// TIA Portal V18 export
ORGANIZATION_BLOCK "Main"   // OB123, FBD, ProgramCycle
TITLE = "Main Program Sweep (Cycle)"
{ S7_Optimized_Access := 'TRUE' }
VERSION : 0.1
// stored: AutoNumber true, IsIECCheckEnabled false, SetENOAutomatically false
   VAR_INPUT
      Initial_Call : Bool;   // Initial call of this OB
      Remanence : Bool;   // =True, if remanent data are available
   END_VAR
BEGIN

REGION Network 1 (SCL): HSSR_019 SOURCE SELECTION

   "Source_select_H/SSR_019_DB".START := "H/SSR_019_START";
   "Source_select_H/SSR_019_DB".SP := "H/SSR_019_SP";
   "Source_select_H/SSR_019_DB".PV := "H/SSR_019_TT01_PV";
   "Source_select_H/SSR_019_DB".COUNTER_SP := "H/SSR_019_ALERT_SP";
   "Source_select_H/SSR_019_DB".CHW_CT_SP := "H/SSR_019_CHBr_RT_SP";
   "Source_select_H/SSR_019_DB".CT_HW_SP := "H/SSR_019_RT_HW_SP";
   "Source_select_H/SSR_019_DB".HW_STEAM_SP := "H/SSR_019_HW_STEAM_SP";
   "Source_select_H/SSR_019_DB".CT_CHW_SP := "H/SSR_019_RT_CHBr_SP";

   "H/SSR_019_SOURCE_SEL" := "Source_select_H/SSR_019_DB".SOURCE_SEL;
END_REGION

REGION Network 2 (SCL): HSSR_019 UTILITY PID

   "Utility_PID_DB".AM := "H/SSR_019_AM";
   "Utility_PID_DB".START := "H/SSR_019_START";
   "Utility_PID_DB".SP := "H/SSR_019_SP";
   "Utility_PID_DB".PV := "H/SSR_019_TT01_PV";
   "Utility_PID_DB".TIME := "H/SSR_019_TIME_SP";
   "Utility_PID_DB".P := "H/SSR_019_KP";
   "Utility_PID_DB".I := "H/SSR_019_TI";
   "Utility_PID_DB".JAC_IN := "H/SSR_019_TT02_PV";
   "Utility_PID_DB".SOURCE_SEL := "Source_select_H/SSR_019_DB".SOURCE_SEL;
   "Utility_PID_DB".MAN_OUT := "H/SSR_019_CV02_MANOUT";
   "Utility_PID_DB".STEAM_MAN_OUT := "H/SSR_019_CV01_MANOUT";
   "Utility_PID_DB".AIR_XV_OPN := "H/SSR_019_XV10_CMD";
   "Utility_PID_DB".BYP_XV_OPN := "H/SSR_019_XV05_CMD";
   "Utility_PID_DB".VENT_OPN := "H/SSR_019_XV06_CMD";
   "Utility_PID_DB".CONDENSATE_XV_OPN := "H/SSR_019_XV12_CMD";
   "Utility_PID_DB".DRAIN_XV_OPN := "H/SSR_019_XV13_CMD";
   "Utility_PID_DB".CONTROL_MODE := 1;

   "H/SSR_019_START_PV" := "Utility_PID_DB".START_PV;
   "H/SSR_019_CV02_SCVOUT" := "Utility_PID_DB".SCVOUT;
   "H/SSR_019_CV02_CVOUT" := "Utility_PID_DB".CVOUT;
   "H/SSR_019_CV01_SCVOUT" := "Utility_PID_DB".STEAM_SCVOUT;
   "H/SSR_019_CV01_CVOUT" := "Utility_PID_DB".STEAM_CVOUT;
   "H/SSR_019_RUN_MIN" := "Utility_PID_DB".RUN_MIN;
END_REGION

REGION Network 3 (SCL): HSSR_019 UTILITY SELECTION

   "Utility_selection_DB".utl_type :=  "Source_select_H/SSR_019_DB".SOURCE_SEL;
   "Utility_selection_DB".chws_cfb :="SIM_VALVE"."H/SSR_019_XV01_CLOSEFB" ;
   "Utility_selection_DB".chws_ofb := "SIM_VALVE"."H/SSR_019_XV01_OPENFB";
   "Utility_selection_DB".cws_cfb := "SIM_VALVE"."H/SSR_019_XV02_CLOSEFB";
   "Utility_selection_DB".cws_ofb := "SIM_VALVE"."H/SSR_019_XV02_OPENFB";
   "Utility_selection_DB".hws_cfb := "SIM_VALVE"."H/SSR_019_XV03_CLOSEFB";
   "Utility_selection_DB".hws_ofb := "SIM_VALVE"."H/SSR_019_XV03_OPENFB";
   "Utility_selection_DB".chwr_cfb := "SIM_VALVE"."H/SSR_019_XV07_CLOSEFB";
   "Utility_selection_DB".chwr_ofb := "SIM_VALVE"."H/SSR_019_XV07_OPENFB";
   "Utility_selection_DB".cwr_cfb := "SIM_VALVE"."H/SSR_019_XV08_CLOSEFB";
   "Utility_selection_DB".cwr_ofb := "SIM_VALVE"."H/SSR_019_XV08_OPENFB";
   "Utility_selection_DB".hwr_cfb := "SIM_VALVE"."H/SSR_019_XV09_CLOSEFB";
   "Utility_selection_DB".hwr_ofb := "SIM_VALVE"."H/SSR_019_XV09_OPENFB";
   "Utility_selection_DB".scv_ofb := "SIM_VALVE"."H/SSR_019_XV11_OPENFB";
   "Utility_selection_DB".cond_cfb := "SIM_VALVE"."H/SSR_019_XV12_CLOSEFB";
   "Utility_selection_DB".cond_ofb := "SIM_VALVE"."H/SSR_019_XV12_OPENFB";
   "Utility_selection_DB".dr_cfb := "SIM_VALVE"."H/SSR_019_XV13_CLOSEFB";
   "Utility_selection_DB".dr_ofb := "SIM_VALVE"."H/SSR_019_XV13_OPENFB";
   "Utility_selection_DB".as_cfb := "SIM_VALVE"."H/SSR_019_XV10_CLOSEFB";
   "Utility_selection_DB".as_ofb := "SIM_VALVE"."H/SSR_019_XV10_OPENFB";
   "Utility_selection_DB".av_cfb := "SIM_VALVE"."H/SSR_019_XV06_CLOSEFB";
   "Utility_selection_DB".av_ofb := "SIM_VALVE"."H/SSR_019_XV06_OPENFB";
   "Utility_selection_DB".utl_bit := "H/SSR_019_START";
   "Utility_selection_DB".control.%X1 := "H/SSR_019_AM";
   "Utility_selection_DB".control.%X2 := "H/SSR_019_START";
   "Utility_selection_DB".times[0] := "H/SSR_019_FLUSH_TIME_SP";
   "Utility_selection_DB".times[1] := "H/SSR_019_VENT_TIME_SP";
   "Utility_selection_DB".times[2] := "H/SSR_019_CONDENSATE_TIME_SP";
   "Utility_selection_DB".control.%X0   := "H/SSR_019_HOLD";
   "Utility_selection_DB".control.%X6 := "H/SSR_019_EMSTOP";
   "Utility_selection_DB".byp_cfb := "SIM_VALVE"."H/SSR_019_XV05_CLOSEFB";
   "Utility_selection_DB".byp_ofb := "SIM_VALVE"."H/SSR_019_XV05_OPENFB";
   "H/SSR_019_XV01_CMD" := "Utility_selection_DB".chws_cmd;
   "H/SSR_019_XV02_CMD" := "Utility_selection_DB".cws_cmd;
   "H/SSR_019_XV03_CMD" := "Utility_selection_DB".hws_cmd;
   "H/SSR_019_XV07_CMD" := "Utility_selection_DB".chwr_cmd;
   "H/SSR_019_XV08_CMD" := "Utility_selection_DB".cwr_cmd;
   "H/SSR_019_XV09_CMD" := "Utility_selection_DB".hwr_cmd;
   "H/SSR_019_XV11_CMD" := "Utility_selection_DB".scv_cmd;
   "H/SSR_019_XV12_CMD" := "Utility_selection_DB".cond_cmd;
   "H/SSR_019_XV13_CMD" := "Utility_selection_DB".dr_cmd;
   "H/SSR_019_XV10_CMD" := "Utility_selection_DB".as_cmd;
   "H/SSR_019_XV05_CMD" := "Utility_selection_DB".byp_cmd;
   "H/SSR_019_XV06_CMD" := "Utility_selection_DB".av_cmd;
   "H/SSR_019_FLUSH_RUN_TIME" := "Utility_selection_DB".flush_time;
   "H/SSR_019_CONDENSATE_RUN_TIME" := "Utility_selection_DB".drine_time;
   "H/SSR_019_VENT_RUN_TIME" := "Utility_selection_DB".vent_time;
   "H/SSR_019_Flush_CMP" := "Utility_selection_DB".status.%X2;
   "H/SSR_019_Vent_CMP" := "Utility_selection_DB".status.%X3;
   "H/SSR_019_Cond_CMP" := "Utility_selection_DB".status.%X4;
END_REGION

REGION Network 4: HSSR_019_Pre checks
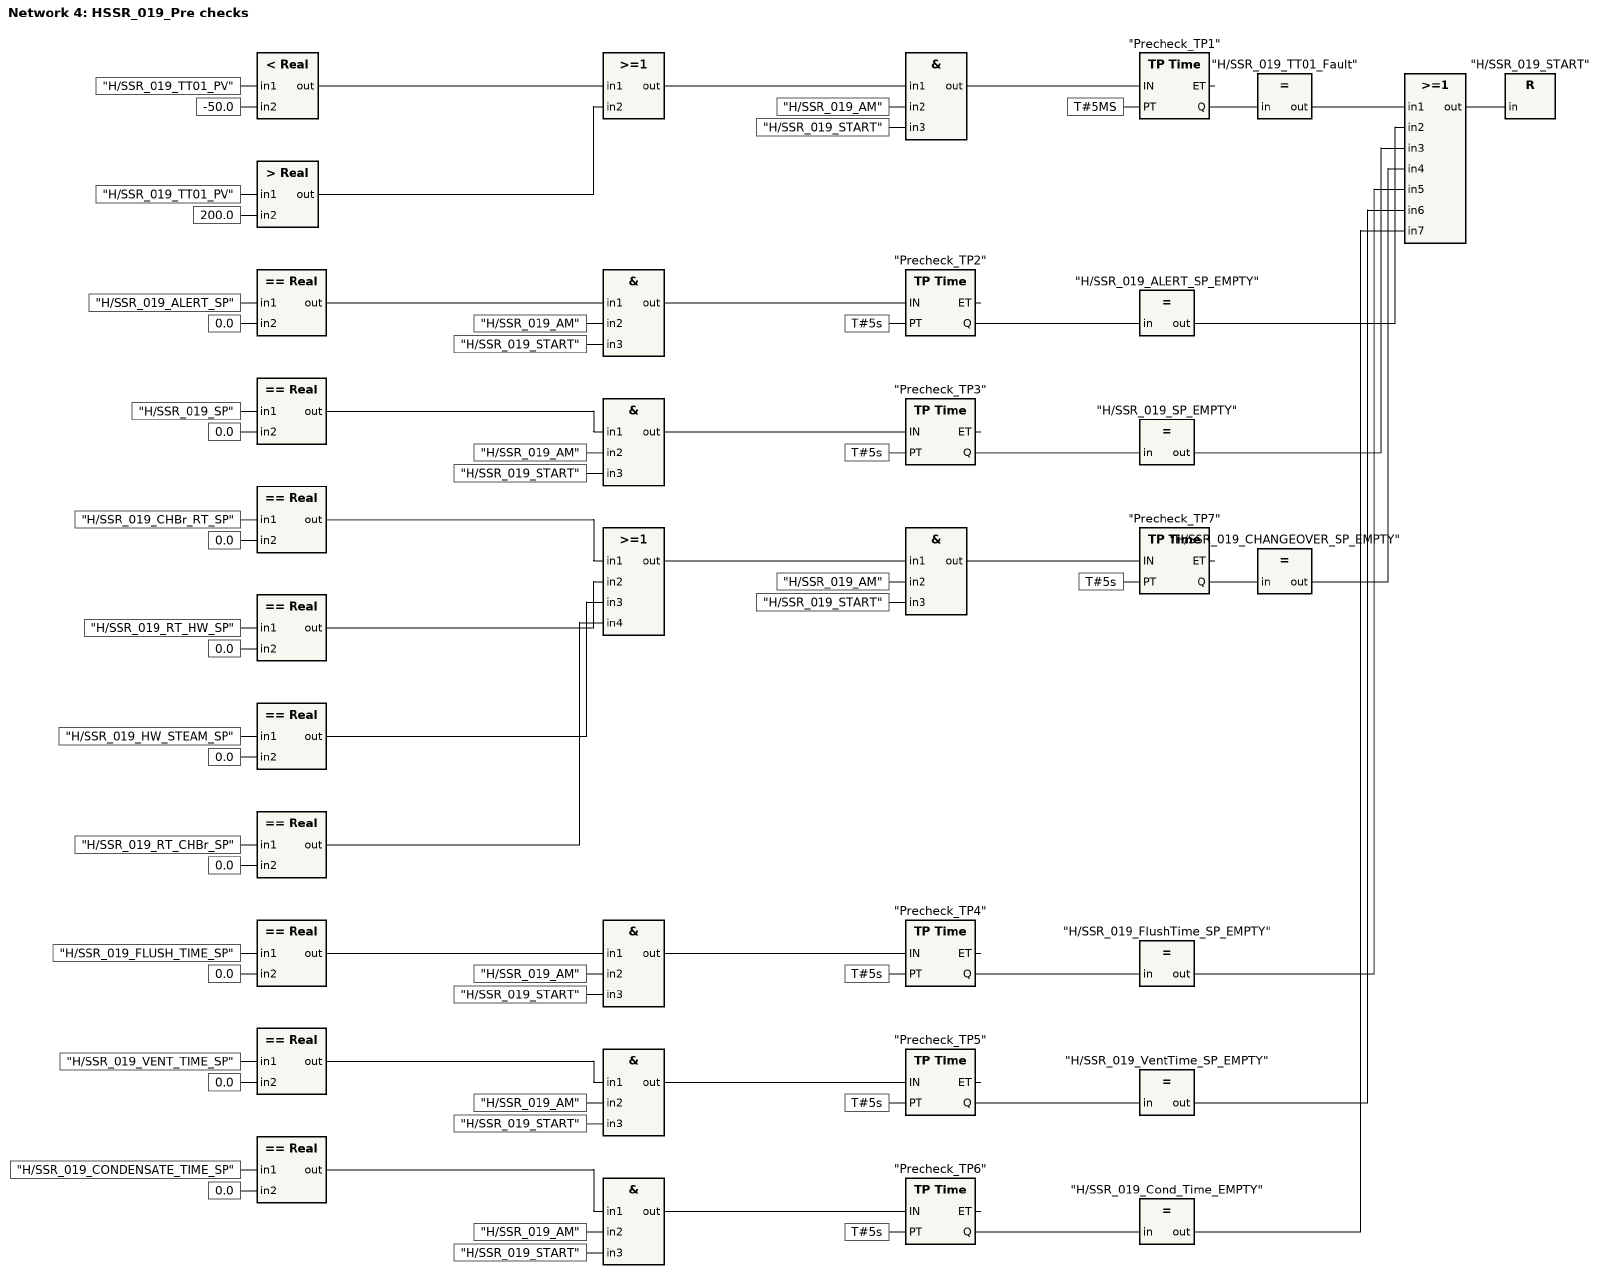
   "Precheck_TP1".TP(IN := (("H/SSR_019_TT01_PV" < (-50.0)) OR ("H/SSR_019_TT01_PV" > 200.0)) AND "H/SSR_019_AM" AND "H/SSR_019_START",
                     PT := T#5MS);
   "H/SSR_019_TT01_Fault" := "Precheck_TP1".Q;
   "Precheck_TP2".TP(IN := ("H/SSR_019_ALERT_SP" = 0.0) AND "H/SSR_019_AM" AND "H/SSR_019_START", PT := T#5s);
   "H/SSR_019_ALERT_SP_EMPTY" := "Precheck_TP2".Q;
   "Precheck_TP3".TP(IN := ("H/SSR_019_SP" = 0.0) AND "H/SSR_019_AM" AND "H/SSR_019_START", PT := T#5s);
   "H/SSR_019_SP_EMPTY" := "Precheck_TP3".Q;
   "Precheck_TP7".TP(IN := (("H/SSR_019_CHBr_RT_SP" = 0.0) OR ("H/SSR_019_RT_HW_SP" = 0.0) OR ("H/SSR_019_HW_STEAM_SP" = 0.0) OR ("H/SSR_019_RT_CHBr_SP" = 0.0)) AND "H/SSR_019_AM" AND "H/SSR_019_START",
                     PT := T#5s);
   "H/SSR_019_CHANGEOVER_SP_EMPTY" := "Precheck_TP7".Q;
   "Precheck_TP4".TP(IN := ("H/SSR_019_FLUSH_TIME_SP" = 0.0) AND "H/SSR_019_AM" AND "H/SSR_019_START",
                     PT := T#5s);
   "H/SSR_019_FlushTime_SP_EMPTY" := "Precheck_TP4".Q;
   "Precheck_TP5".TP(IN := ("H/SSR_019_VENT_TIME_SP" = 0.0) AND "H/SSR_019_AM" AND "H/SSR_019_START",
                     PT := T#5s);
   "H/SSR_019_VentTime_SP_EMPTY" := "Precheck_TP5".Q;
   "Precheck_TP6".TP(IN := ("H/SSR_019_CONDENSATE_TIME_SP" = 0.0) AND "H/SSR_019_AM" AND "H/SSR_019_START",
                     PT := T#5s);
   "H/SSR_019_Cond_Time_EMPTY" := "Precheck_TP6".Q;
   IF "Precheck_TP1".Q OR "Precheck_TP2".Q OR "Precheck_TP3".Q OR "Precheck_TP7".Q OR "Precheck_TP4".Q OR "Precheck_TP5".Q OR "Precheck_TP6".Q THEN
       "H/SSR_019_START" := FALSE;
   END_IF;
END_REGION

REGION Network 5: H/SSR_019Valves
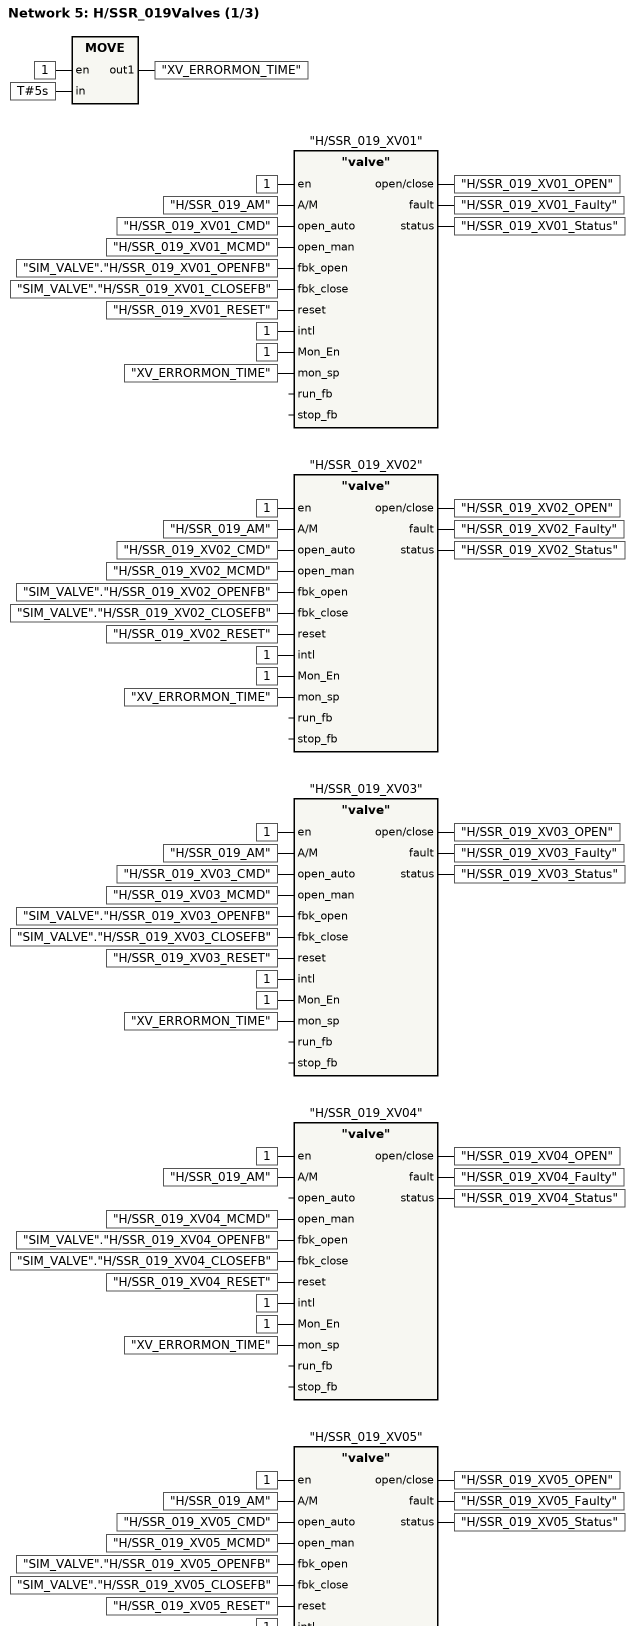
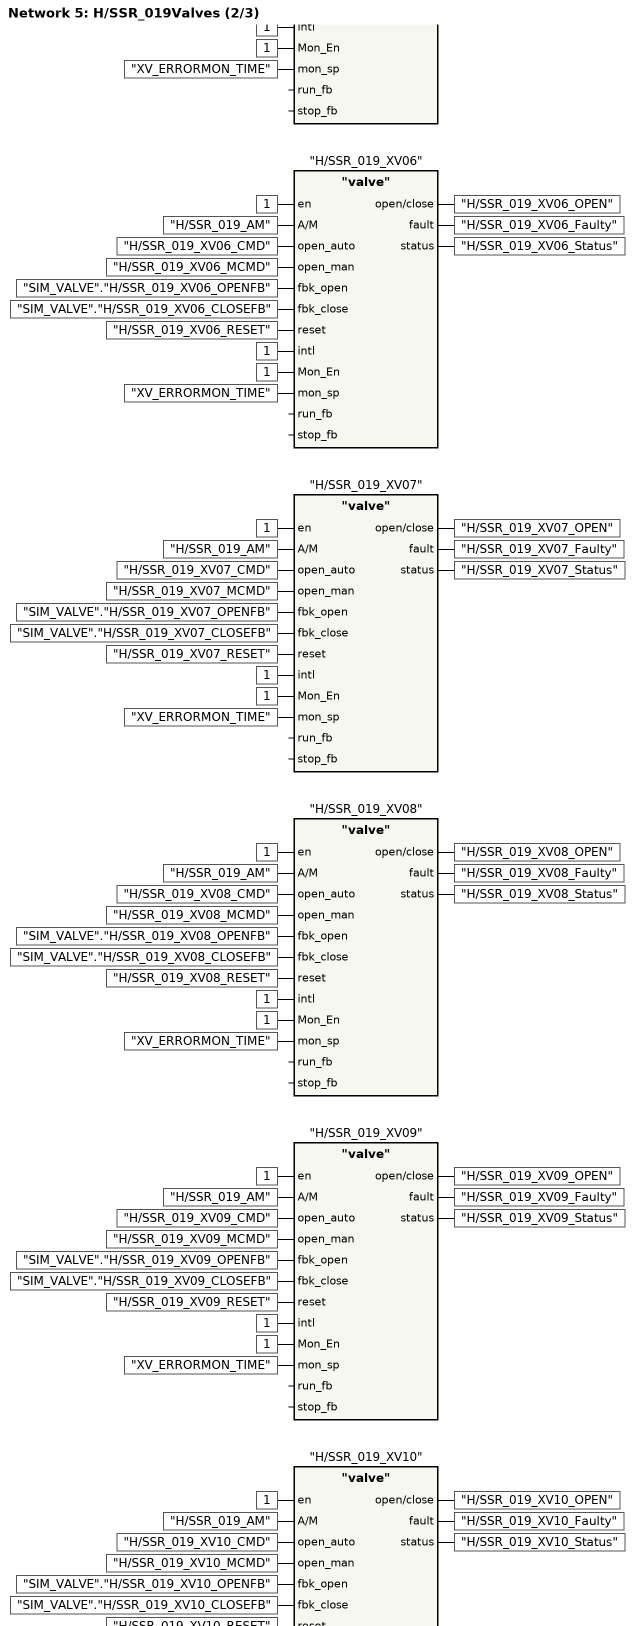
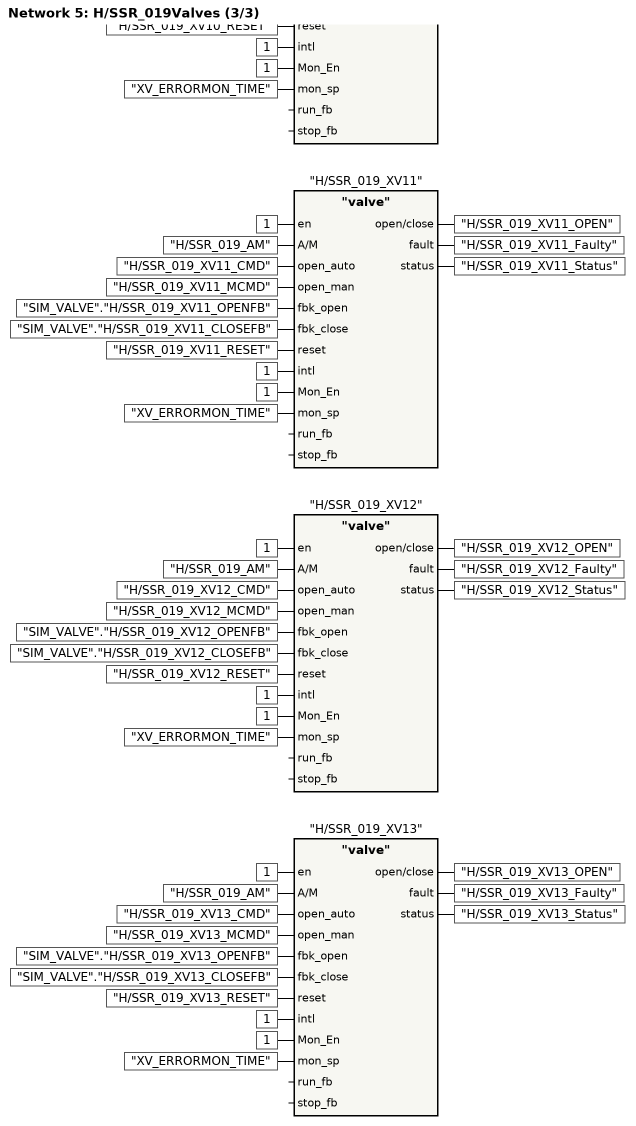
   IF 1 THEN
       "XV_ERRORMON_TIME" := T#5s;
       "H/SSR_019_XV01"("A/M" := "H/SSR_019_AM",   // "valve"
                        open_auto := "H/SSR_019_XV01_CMD",
                        open_man := "H/SSR_019_XV01_MCMD",
                        fbk_open := "SIM_VALVE"."H/SSR_019_XV01_OPENFB",
                        fbk_close := "SIM_VALVE"."H/SSR_019_XV01_CLOSEFB",
                        reset := "H/SSR_019_XV01_RESET",
                        intl := 1,
                        Mon_En := 1,
                        mon_sp := "XV_ERRORMON_TIME",
                        "open/close" => "H/SSR_019_XV01_OPEN",
                        fault => "H/SSR_019_XV01_Faulty",
                        status => "H/SSR_019_XV01_Status");
       "H/SSR_019_XV02"("A/M" := "H/SSR_019_AM",   // "valve"
                        open_auto := "H/SSR_019_XV02_CMD",
                        open_man := "H/SSR_019_XV02_MCMD",
                        fbk_open := "SIM_VALVE"."H/SSR_019_XV02_OPENFB",
                        fbk_close := "SIM_VALVE"."H/SSR_019_XV02_CLOSEFB",
                        reset := "H/SSR_019_XV02_RESET",
                        intl := 1,
                        Mon_En := 1,
                        mon_sp := "XV_ERRORMON_TIME",
                        "open/close" => "H/SSR_019_XV02_OPEN",
                        fault => "H/SSR_019_XV02_Faulty",
                        status => "H/SSR_019_XV02_Status");
       "H/SSR_019_XV03"("A/M" := "H/SSR_019_AM",   // "valve"
                        open_auto := "H/SSR_019_XV03_CMD",
                        open_man := "H/SSR_019_XV03_MCMD",
                        fbk_open := "SIM_VALVE"."H/SSR_019_XV03_OPENFB",
                        fbk_close := "SIM_VALVE"."H/SSR_019_XV03_CLOSEFB",
                        reset := "H/SSR_019_XV03_RESET",
                        intl := 1,
                        Mon_En := 1,
                        mon_sp := "XV_ERRORMON_TIME",
                        "open/close" => "H/SSR_019_XV03_OPEN",
                        fault => "H/SSR_019_XV03_Faulty",
                        status => "H/SSR_019_XV03_Status");
       "H/SSR_019_XV04"("A/M" := "H/SSR_019_AM",   // "valve"
                        open_man := "H/SSR_019_XV04_MCMD",
                        fbk_open := "SIM_VALVE"."H/SSR_019_XV04_OPENFB",
                        fbk_close := "SIM_VALVE"."H/SSR_019_XV04_CLOSEFB",
                        reset := "H/SSR_019_XV04_RESET",
                        intl := 1,
                        Mon_En := 1,
                        mon_sp := "XV_ERRORMON_TIME",
                        "open/close" => "H/SSR_019_XV04_OPEN",
                        fault => "H/SSR_019_XV04_Faulty",
                        status => "H/SSR_019_XV04_Status");
       "H/SSR_019_XV05"("A/M" := "H/SSR_019_AM",   // "valve"
                        open_auto := "H/SSR_019_XV05_CMD",
                        open_man := "H/SSR_019_XV05_MCMD",
                        fbk_open := "SIM_VALVE"."H/SSR_019_XV05_OPENFB",
                        fbk_close := "SIM_VALVE"."H/SSR_019_XV05_CLOSEFB",
                        reset := "H/SSR_019_XV05_RESET",
                        intl := 1,
                        Mon_En := 1,
                        mon_sp := "XV_ERRORMON_TIME",
                        "open/close" => "H/SSR_019_XV05_OPEN",
                        fault => "H/SSR_019_XV05_Faulty",
                        status => "H/SSR_019_XV05_Status");
       "H/SSR_019_XV06"("A/M" := "H/SSR_019_AM",   // "valve"
                        open_auto := "H/SSR_019_XV06_CMD",
                        open_man := "H/SSR_019_XV06_MCMD",
                        fbk_open := "SIM_VALVE"."H/SSR_019_XV06_OPENFB",
                        fbk_close := "SIM_VALVE"."H/SSR_019_XV06_CLOSEFB",
                        reset := "H/SSR_019_XV06_RESET",
                        intl := 1,
                        Mon_En := 1,
                        mon_sp := "XV_ERRORMON_TIME",
                        "open/close" => "H/SSR_019_XV06_OPEN",
                        fault => "H/SSR_019_XV06_Faulty",
                        status => "H/SSR_019_XV06_Status");
       "H/SSR_019_XV07"("A/M" := "H/SSR_019_AM",   // "valve"
                        open_auto := "H/SSR_019_XV07_CMD",
                        open_man := "H/SSR_019_XV07_MCMD",
                        fbk_open := "SIM_VALVE"."H/SSR_019_XV07_OPENFB",
                        fbk_close := "SIM_VALVE"."H/SSR_019_XV07_CLOSEFB",
                        reset := "H/SSR_019_XV07_RESET",
                        intl := 1,
                        Mon_En := 1,
                        mon_sp := "XV_ERRORMON_TIME",
                        "open/close" => "H/SSR_019_XV07_OPEN",
                        fault => "H/SSR_019_XV07_Faulty",
                        status => "H/SSR_019_XV07_Status");
       "H/SSR_019_XV08"("A/M" := "H/SSR_019_AM",   // "valve"
                        open_auto := "H/SSR_019_XV08_CMD",
                        open_man := "H/SSR_019_XV08_MCMD",
                        fbk_open := "SIM_VALVE"."H/SSR_019_XV08_OPENFB",
                        fbk_close := "SIM_VALVE"."H/SSR_019_XV08_CLOSEFB",
                        reset := "H/SSR_019_XV08_RESET",
                        intl := 1,
                        Mon_En := 1,
                        mon_sp := "XV_ERRORMON_TIME",
                        "open/close" => "H/SSR_019_XV08_OPEN",
                        fault => "H/SSR_019_XV08_Faulty",
                        status => "H/SSR_019_XV08_Status");
       "H/SSR_019_XV09"("A/M" := "H/SSR_019_AM",   // "valve"
                        open_auto := "H/SSR_019_XV09_CMD",
                        open_man := "H/SSR_019_XV09_MCMD",
                        fbk_open := "SIM_VALVE"."H/SSR_019_XV09_OPENFB",
                        fbk_close := "SIM_VALVE"."H/SSR_019_XV09_CLOSEFB",
                        reset := "H/SSR_019_XV09_RESET",
                        intl := 1,
                        Mon_En := 1,
                        mon_sp := "XV_ERRORMON_TIME",
                        "open/close" => "H/SSR_019_XV09_OPEN",
                        fault => "H/SSR_019_XV09_Faulty",
                        status => "H/SSR_019_XV09_Status");
       "H/SSR_019_XV10"("A/M" := "H/SSR_019_AM",   // "valve"
                        open_auto := "H/SSR_019_XV10_CMD",
                        open_man := "H/SSR_019_XV10_MCMD",
                        fbk_open := "SIM_VALVE"."H/SSR_019_XV10_OPENFB",
                        fbk_close := "SIM_VALVE"."H/SSR_019_XV10_CLOSEFB",
                        reset := "H/SSR_019_XV10_RESET",
                        intl := 1,
                        Mon_En := 1,
                        mon_sp := "XV_ERRORMON_TIME",
                        "open/close" => "H/SSR_019_XV10_OPEN",
                        fault => "H/SSR_019_XV10_Faulty",
                        status => "H/SSR_019_XV10_Status");
       "H/SSR_019_XV11"("A/M" := "H/SSR_019_AM",   // "valve"
                        open_auto := "H/SSR_019_XV11_CMD",
                        open_man := "H/SSR_019_XV11_MCMD",
                        fbk_open := "SIM_VALVE"."H/SSR_019_XV11_OPENFB",
                        fbk_close := "SIM_VALVE"."H/SSR_019_XV11_CLOSEFB",
                        reset := "H/SSR_019_XV11_RESET",
                        intl := 1,
                        Mon_En := 1,
                        mon_sp := "XV_ERRORMON_TIME",
                        "open/close" => "H/SSR_019_XV11_OPEN",
                        fault => "H/SSR_019_XV11_Faulty",
                        status => "H/SSR_019_XV11_Status");
       "H/SSR_019_XV12"("A/M" := "H/SSR_019_AM",   // "valve"
                        open_auto := "H/SSR_019_XV12_CMD",
                        open_man := "H/SSR_019_XV12_MCMD",
                        fbk_open := "SIM_VALVE"."H/SSR_019_XV12_OPENFB",
                        fbk_close := "SIM_VALVE"."H/SSR_019_XV12_CLOSEFB",
                        reset := "H/SSR_019_XV12_RESET",
                        intl := 1,
                        Mon_En := 1,
                        mon_sp := "XV_ERRORMON_TIME",
                        "open/close" => "H/SSR_019_XV12_OPEN",
                        fault => "H/SSR_019_XV12_Faulty",
                        status => "H/SSR_019_XV12_Status");
       "H/SSR_019_XV13"("A/M" := "H/SSR_019_AM",   // "valve"
                        open_auto := "H/SSR_019_XV13_CMD",
                        open_man := "H/SSR_019_XV13_MCMD",
                        fbk_open := "SIM_VALVE"."H/SSR_019_XV13_OPENFB",
                        fbk_close := "SIM_VALVE"."H/SSR_019_XV13_CLOSEFB",
                        reset := "H/SSR_019_XV13_RESET",
                        intl := 1,
                        Mon_En := 1,
                        mon_sp := "XV_ERRORMON_TIME",
                        "open/close" => "H/SSR_019_XV13_OPEN",
                        fault => "H/SSR_019_XV13_Faulty",
                        status => "H/SSR_019_XV13_Status");
   END_IF;
END_REGION

REGION Network 6: AI_H/SSR_019_ Reading
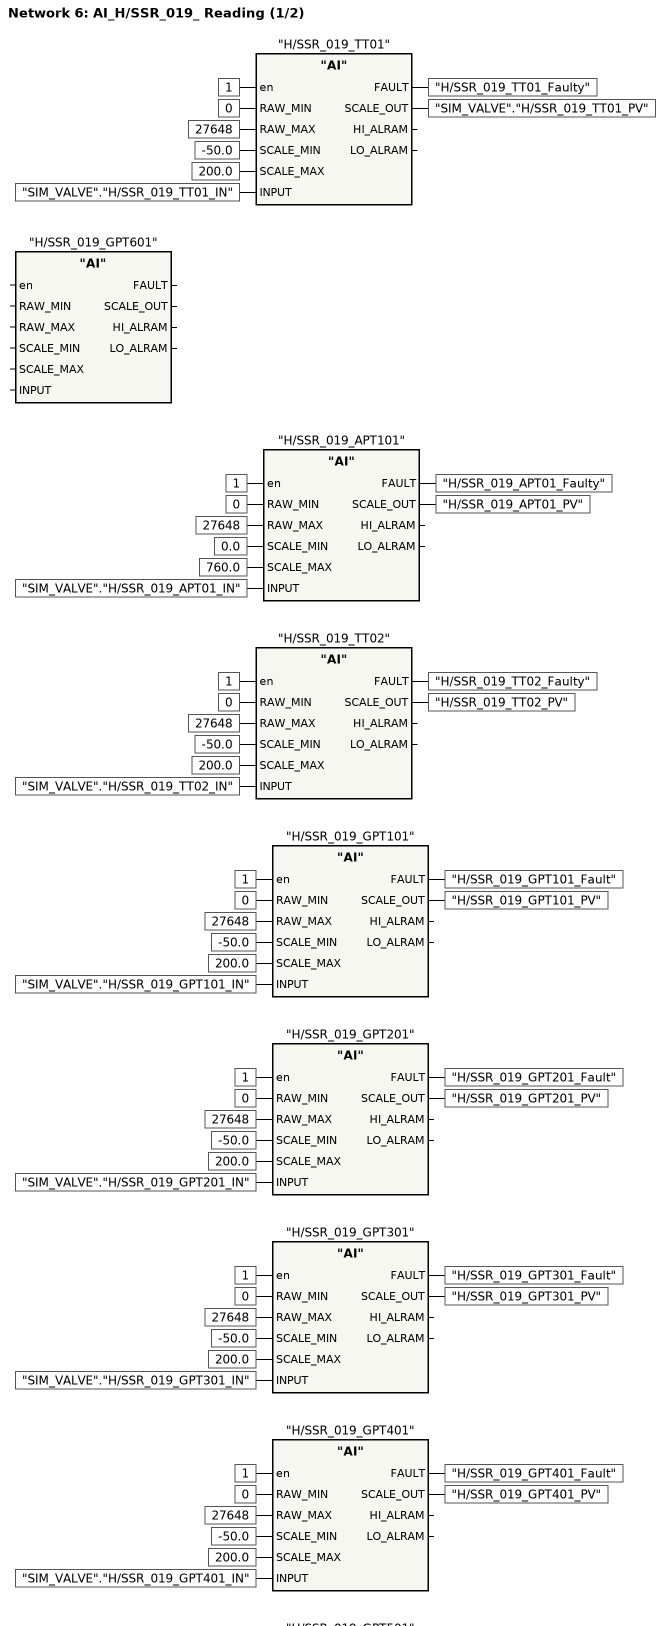
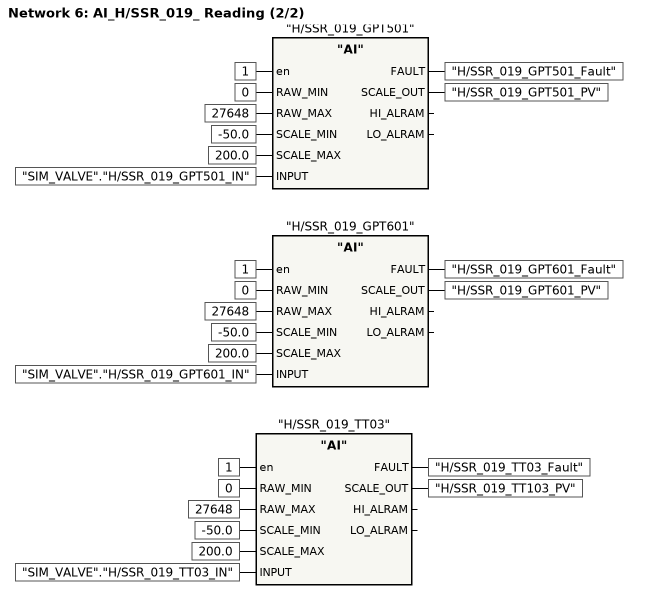
   IF 1 THEN
       "H/SSR_019_TT01"(RAW_MIN := 0,   // "AI"
                        RAW_MAX := 27648,
                        SCALE_MIN := -50.0,
                        SCALE_MAX := 200.0,
                        INPUT := "SIM_VALVE"."H/SSR_019_TT01_IN",
                        FAULT => "H/SSR_019_TT01_Faulty",
                        SCALE_OUT => "SIM_VALVE"."H/SSR_019_TT01_PV");
   END_IF;
   "H/SSR_019_GPT601"();   // "AI"
   IF 1 THEN
       "H/SSR_019_APT101"(RAW_MIN := 0,   // "AI"
                          RAW_MAX := 27648,
                          SCALE_MIN := 0.0,
                          SCALE_MAX := 760.0,
                          INPUT := "SIM_VALVE"."H/SSR_019_APT01_IN",
                          FAULT => "H/SSR_019_APT01_Faulty",
                          SCALE_OUT => "H/SSR_019_APT01_PV");
       "H/SSR_019_TT02"(RAW_MIN := 0,   // "AI"
                        RAW_MAX := 27648,
                        SCALE_MIN := -50.0,
                        SCALE_MAX := 200.0,
                        INPUT := "SIM_VALVE"."H/SSR_019_TT02_IN",
                        FAULT => "H/SSR_019_TT02_Faulty",
                        SCALE_OUT => "H/SSR_019_TT02_PV");
       "H/SSR_019_GPT101"(RAW_MIN := 0,   // "AI"
                          RAW_MAX := 27648,
                          SCALE_MIN := -50.0,
                          SCALE_MAX := 200.0,
                          INPUT := "SIM_VALVE"."H/SSR_019_GPT101_IN",
                          FAULT => "H/SSR_019_GPT101_Fault",
                          SCALE_OUT => "H/SSR_019_GPT101_PV");
       "H/SSR_019_GPT201"(RAW_MIN := 0,   // "AI"
                          RAW_MAX := 27648,
                          SCALE_MIN := -50.0,
                          SCALE_MAX := 200.0,
                          INPUT := "SIM_VALVE"."H/SSR_019_GPT201_IN",
                          FAULT => "H/SSR_019_GPT201_Fault",
                          SCALE_OUT => "H/SSR_019_GPT201_PV");
       "H/SSR_019_GPT301"(RAW_MIN := 0,   // "AI"
                          RAW_MAX := 27648,
                          SCALE_MIN := -50.0,
                          SCALE_MAX := 200.0,
                          INPUT := "SIM_VALVE"."H/SSR_019_GPT301_IN",
                          FAULT => "H/SSR_019_GPT301_Fault",
                          SCALE_OUT => "H/SSR_019_GPT301_PV");
       "H/SSR_019_GPT401"(RAW_MIN := 0,   // "AI"
                          RAW_MAX := 27648,
                          SCALE_MIN := -50.0,
                          SCALE_MAX := 200.0,
                          INPUT := "SIM_VALVE"."H/SSR_019_GPT401_IN",
                          FAULT => "H/SSR_019_GPT401_Fault",
                          SCALE_OUT => "H/SSR_019_GPT401_PV");
       "H/SSR_019_GPT501"(RAW_MIN := 0,   // "AI"
                          RAW_MAX := 27648,
                          SCALE_MIN := -50.0,
                          SCALE_MAX := 200.0,
                          INPUT := "SIM_VALVE"."H/SSR_019_GPT501_IN",
                          FAULT => "H/SSR_019_GPT501_Fault",
                          SCALE_OUT => "H/SSR_019_GPT501_PV");
       "H/SSR_019_GPT601"(RAW_MIN := 0,   // "AI"
                          RAW_MAX := 27648,
                          SCALE_MIN := -50.0,
                          SCALE_MAX := 200.0,
                          INPUT := "SIM_VALVE"."H/SSR_019_GPT601_IN",
                          FAULT => "H/SSR_019_GPT601_Fault",
                          SCALE_OUT => "H/SSR_019_GPT601_PV");
       "H/SSR_019_TT03"(RAW_MIN := 0,   // "AI"
                        RAW_MAX := 27648,
                        SCALE_MIN := -50.0,
                        SCALE_MAX := 200.0,
                        INPUT := "SIM_VALVE"."H/SSR_019_TT03_IN",
                        FAULT => "H/SSR_019_TT03_Fault",
                        SCALE_OUT => "H/SSR_019_TT103_PV");
   END_IF;
END_REGION

REGION Network 7: Agitaor
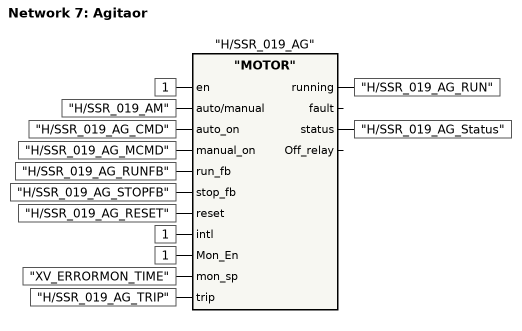
   IF 1 THEN
       "H/SSR_019_AG"("auto/manual" := "H/SSR_019_AM",   // "MOTOR"
                      auto_on := "H/SSR_019_AG_CMD",
                      manual_on := "H/SSR_019_AG_MCMD",
                      run_fb := "H/SSR_019_AG_RUNFB",
                      stop_fb := "H/SSR_019_AG_STOPFB",
                      reset := "H/SSR_019_AG_RESET",
                      intl := 1,
                      Mon_En := 1,
                      mon_sp := "XV_ERRORMON_TIME",
                      trip := "H/SSR_019_AG_TRIP",
                      running => "H/SSR_019_AG_RUN",
                      status => "H/SSR_019_AG_Status");
   END_IF;
END_REGION

REGION Network 8: H/SSR_019 GLOBAL RESET
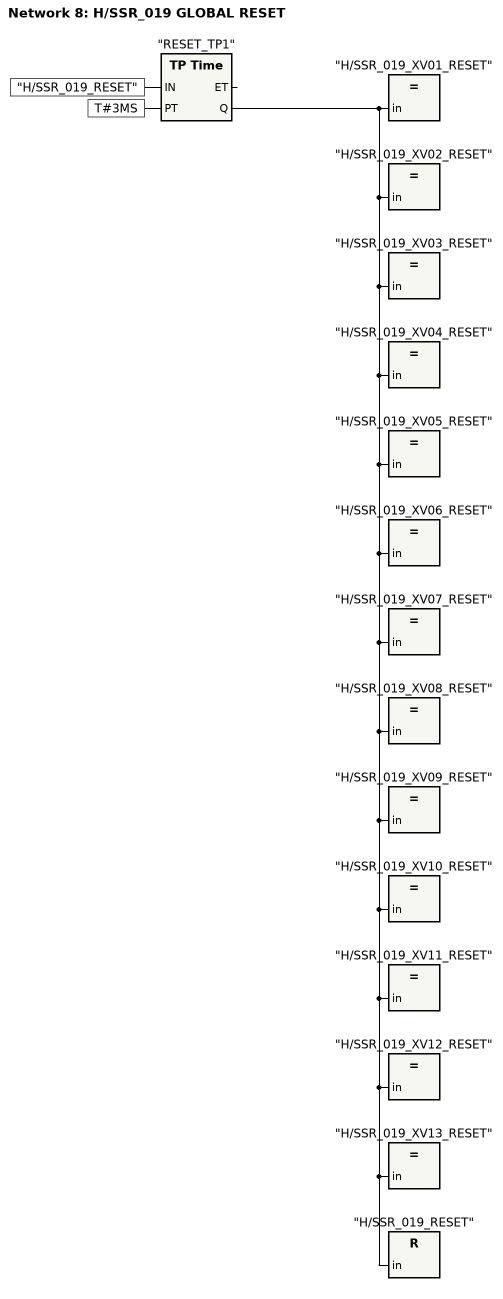
   "RESET_TP1".TP(IN := "H/SSR_019_RESET", PT := T#3MS);
   "H/SSR_019_XV01_RESET" := "RESET_TP1".Q;
   "H/SSR_019_XV02_RESET" := "RESET_TP1".Q;
   "H/SSR_019_XV03_RESET" := "RESET_TP1".Q;
   "H/SSR_019_XV04_RESET" := "RESET_TP1".Q;
   "H/SSR_019_XV05_RESET" := "RESET_TP1".Q;
   "H/SSR_019_XV06_RESET" := "RESET_TP1".Q;
   "H/SSR_019_XV07_RESET" := "RESET_TP1".Q;
   "H/SSR_019_XV08_RESET" := "RESET_TP1".Q;
   "H/SSR_019_XV09_RESET" := "RESET_TP1".Q;
   "H/SSR_019_XV10_RESET" := "RESET_TP1".Q;
   "H/SSR_019_XV11_RESET" := "RESET_TP1".Q;
   "H/SSR_019_XV12_RESET" := "RESET_TP1".Q;
   "H/SSR_019_XV13_RESET" := "RESET_TP1".Q;
   IF "RESET_TP1".Q THEN "H/SSR_019_RESET" := FALSE; END_IF;
END_REGION

REGION Network 9: HOOTER
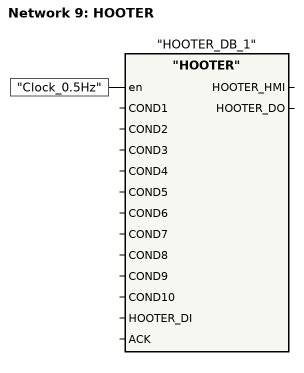
   IF "Clock_0.5Hz" THEN
       "HOOTER_DB_1"();   // "HOOTER"
   END_IF;
END_REGION
END_ORGANIZATION_BLOCK
